TYPE SStrategy :
STRUCT
	State: EStrategyStates;
	
	LoopStrategy: BOOL;
	Steps: ARRAY [ResiConst.ARR_MIN..ResiConst.STRAT_LEN_MAX] OF SStep;
	Transitions: ARRAY [ResiConst.ARR_MIN..ResiConst.STRAT_LEN_MAX] OF STransition;
	
	IsMaster: BOOL;
	NumPartners: UINT;
END_STRUCT
END_TYPE

(* stored: Version 1.1.0.1
   DUT SStrategy: Id {919936fe-6b28-430a-ba3e-fc9c4d6db738} *)
